FUNCTION TryConvert_DWORD_TO_INT : BOOL
VAR_INPUT
	in : DWORD;
	out : REFERENCE TO INT;
END_VAR

IF in > DatatypeLimits.MAX_VALUE_OF_DWORD_WHICH_CAN_BE_HELD_IN_A_INT THEN
	RETURN;
END_IF

out := DWORD_TO_INT(in);
TryConvert_DWORD_TO_INT := TRUE;

END_FUNCTION

(* stored: Version 1.1.0.1, ProductVersion 3.1.4024.12
   POU TryConvert_DWORD_TO_INT: Id {7afa1160-ffd5-46b7-a0ea-80d130f00a9a}, SpecialFunc None *)
